{attribute addProperty BoxType "IODEVICETYPE_ETHERCATPROT"}
{attribute addProperty Id "Beckhoff_EJ1xxxBeckhoff_EJ1xxx_1EC3FDB8968121Beckhoff_EJ2xxxBeckhoff_EJ2xxx_A610010F1792224Beckhoff_EJ3xxxBeckhoff_EJ3xxx_92F483A76082760.25Beckhoff_EJ4xxxBeckhoff_EJ4xxx_9403FF521416177Beckhoff_EJ5xxxBeckhoff_EJ5xxx_9065C16178498Beckhoff_EJ6xxxBeckhoff_EJ6xxx_5DE87ABD1264158Beckhoff_EJ7xxxBeckhoff_EJ7xxx_CCAB573786961087Beckhoff_EJ9xxxBeckhoff_EJ9xxx_158E4C7F992124Beckhoff_EJx9xxBeckhoff_EJx9xx_67C605582896362SyncUnitsSyncUnits_3FA29F3C21627InputsInputs_C75D3FEC1280160OutputsOutputs_47D1E803848106InfoDataInfoData_45F98C5022428"}
{attribute addProperty CRC "3062280204"}
{attribute addProperty SizeInBites "27458"}
{attribute addProperty SizeInBytes "3432.25"}
TYPE EtherCAT_Master_EJxxxx_B686B00C :
STRUCT
	{attribute addProperty Name "Beckhoff_EJ1xxx"}
	Beckhoff_EJ1xxx : Beckhoff_EJ1xxx_1EC3FDB8;
	{attribute addProperty Name "Beckhoff_EJ2xxx"}
	Beckhoff_EJ2xxx : Beckhoff_EJ2xxx_A610010F;
	{attribute addProperty Name "Beckhoff_EJ3xxx"}
	Beckhoff_EJ3xxx : Beckhoff_EJ3xxx_92F483A7;
	{attribute addProperty Name "Beckhoff_EJ4xxx"}
	Beckhoff_EJ4xxx : Beckhoff_EJ4xxx_9403FF52;
	{attribute addProperty Name "Beckhoff_EJ5xxx"}
	Beckhoff_EJ5xxx : Beckhoff_EJ5xxx_9065C161;
	{attribute addProperty Name "Beckhoff_EJ6xxx"}
	Beckhoff_EJ6xxx : Beckhoff_EJ6xxx_5DE87ABD;
	{attribute addProperty Name "Beckhoff_EJ7xxx"}
	Beckhoff_EJ7xxx : Beckhoff_EJ7xxx_CCAB5737;
	{attribute addProperty Name "Beckhoff_EJ9xxx"}
	Beckhoff_EJ9xxx : Beckhoff_EJ9xxx_158E4C7F;
	{attribute addProperty Name "Beckhoff_EJx9xx"}
	Beckhoff_EJx9xx : Beckhoff_EJx9xx_67C60558;
	{attribute addProperty Name "SyncUnits"}
	SyncUnits : SyncUnits_3FA29F3C;
	{attribute addProperty Name "Inputs"}
	Inputs : Inputs_C75D3FEC;
	{attribute addProperty Name "Outputs"}
	Outputs : Outputs_47D1E803;
	{attribute addProperty Name "InfoData"}
	InfoData : InfoData_45F98C50;
END_STRUCT
END_TYPE

(* stored: Version 1.2.0.0, ProductVersion 3.1.4024.9
   DUT EtherCAT_Master_EJxxxx_B686B00C: Id {ec31dede-e00b-4e8e-b545-4c21a958912f} *)
